FUNCTION Sign : LREAL
VAR_INPUT
	in	: LREAL;
END_VAR
VAR
END_VAR

IF in > 0.0 THEN
	Sign := 1.0;
ELSE
	Sign := -1.0;
END_IF

END_FUNCTION

(* stored: Version 1.1.0.1, ProductVersion 3.1.4024.9
   POU Sign: Id {4b830b40-4eaf-45b3-aa8f-37c619dc1cfc}, SpecialFunc None *)
